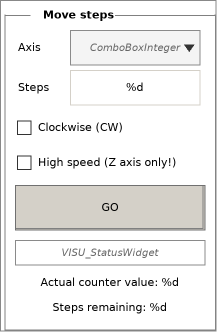
VISUALIZATION VISU_M2MoveSteps  // 217x332
VAR_IN_OUT
	ref_process   : M2MoveStepsProcess;
	ref_procedure : M2MoveStepsProcedure;
    widget : M2MoveStepsWidget;
END_VAR
    Label (40,5 150x20), "Move steps"
    Polyline (115,15) (215,15) (215,330) (5,330) (5,15) (30,15)
    Frame (15,240 190x25)
        shows VISU_StatusWidget(widget := widget.actualStatus)
    ComboBoxInteger (70,30 130x35), variable: ref_process.set.axis, input disabled if: ref_process.statuses.enabledStatus.disabled, text list: 'M2AxesTextList'
    Label (15,30 50x35), "Axis"
    Checkbox (15,145 185x35), "High speed (Z axis only!)", variable: ref_process.set.fast, input disabled if: ref_process.statuses.enabledStatus.disabled
    Button (15,185 190x45), "GO", input disabled if: ref_process.statuses.enabledStatus.disabled
        OnMouseClick: execute { ref_process.do_request := TRUE; }
    Rectangle (15,270 190x25), "Actual counter value: %d", text variable: ref_procedure.actualCounterValue
    Label (15,70 50x35), "Steps"
    Textfield (70,70 130x35), "%d", text variable: ref_process.set.steps, input disabled if: ref_process.statuses.enabledStatus.disabled
        OnMouseClick: write the text variable via VisuDialogs.Numpad, title 'Number of steps to move'
    Checkbox (15,110 195x35), "Clockwise (CW)", variable: ref_process.set.cw, input disabled if: ref_process.statuses.enabledStatus.disabled
    Rectangle (15,295 190x25), "Steps remaining: %d", text variable: ref_procedure.stepsRemaining
END_VISUALIZATION

(* stored: Version 1.1.0.1, ProductVersion 3.1.4019.2
   Visu VISU_M2MoveSteps: Id {57e03ba4-126d-4e77-b1da-7a61fb8ad4d0} *)
